// TIA Portal V16 export
// export: Created 2021-11-12T13:32:04.0416234Z, ExportSetting WithDefaults, DisplayName Totally Integrated Automation Portal, DisplayVersion V16 Update 3, DisplayName TIA Portal Version Control Interface, DisplayVersion V16 Update 2, DisplayName TIA Portal Openness, DisplayVersion V16 Update 3, DisplayName SINAMICS Startdrive Advanced, DisplayVersion V16 Update 5, DisplayName SINAMICS Startdrive G130, G150, S120, S150, SINAMICS MV, S210, DisplayVersion V16 Update 5, DisplayName SINAMICS Startdrive G110M, G120, G120C, G120D, G120P, G115D, DisplayVersion V16 Update 5, DisplayName STEP 7 Professional, DisplayVersion V16 Update 3, DisplayName STEP 7 Safety, DisplayVersion V16, DisplayName WinCC UA Professional, DisplayVersion V16 Update 3
DATA_BLOCK "IDB_Station110"   // DB202
VERSION : 0.1
// stored: AutoNumber true, DBAccessibleFromOPCUA true, InstanceOfName Station 110, InstanceOfType FB
"Station 110"
   // VAR
   //    SF_Alarm1 : "STD_DI_Mon";
   //    SF_Alarm2 { S7_SetPoint := 'True'} : "STD_DI_Mon";
   //    SF_Alarm3 { S7_SetPoint := 'True'} : "STD_DI_Mon";
   //    SF_Alarm4 { S7_SetPoint := 'True'} : "STD_DI_Mon";
   //    SF_Alarm5 { S7_SetPoint := 'True'} : "STD_DI_Mon";
   //    SF_Alarm6 { S7_SetPoint := 'True'} : "STD_DI_Mon";
   //    SF_Alarm7 { S7_SetPoint := 'True'} : "STD_DI_Mon";
   //    SF_Alarm8 { S7_SetPoint := 'True'} : "STD_DI_Mon";
   //    SF_Alarm9 { S7_SetPoint := 'True'} : "STD_DI_Mon";
   //    SF_Alarm10 { S7_SetPoint := 'True'} : "STD_DI_Mon";
   //    SF_Alarm11 { S7_SetPoint := 'True'} : "STD_DI_Mon";
   //    SF_Alarm12 { S7_SetPoint := 'True'} : "STD_DI_Mon";
   //    SF_Alarm13 { S7_SetPoint := 'True'} : "STD_DI_Mon";
   //    SF_Alarm14 { S7_SetPoint := 'True'} : "STD_DI_Mon";
   //    SF_Alarm15 { S7_SetPoint := 'True'} : "STD_DI_Mon";
   //    SF_Alarm16 { S7_SetPoint := 'True'} : "STD_DI_Mon";
   //    SF_Alarm17 { S7_SetPoint := 'True'} : "STD_DI_Mon";
   //    SF_Alarm18 { S7_SetPoint := 'True'} : "STD_DI_Mon";
   //    SF_Alarm19 { S7_SetPoint := 'True'} : "STD_DI_Mon";
   //    SF_Alarm20 { S7_SetPoint := 'True'} : "STD_DI_Mon";
   //    SF_Alarm21 { S7_SetPoint := 'True'} : "STD_DI_Mon";
   //    SF_GL01MA02 { S7_SetPoint := 'True'} : "STD_Drive1";
   //    SF_UH31TA01 { S7_SetPoint := 'True'} : "STD_SERVO_FESTO_CMMT";
   //    SF_UC12TA01 { S7_SetPoint := 'True'} : "STD_Siemens_G120_CU240E_2_PN";
   //    SF_GL01BG05 { S7_SetPoint := 'True'} : "STD_Siemens_MC_Encoder";
   //    SF_GL01MM01 { S7_SetPoint := 'True'} : "STD_Valve2WB";
   //    SF_GM01MM01 { S7_SetPoint := 'True'} : "STD_Valve2WB";
   //    SF_GM01MM02 { S7_SetPoint := 'True'} : "STD_Valve2WB";
   //    SF_GM01MM03 { S7_SetPoint := 'True'} : "STD_Valve2WB";
   //    SF_GM01MM04 { S7_SetPoint := 'True'} : "STD_Valve2WB";
   //    SS_Edge : Array[0..9] of Bool;
   //    SF_TON_MeasDelay { S7_SetPoint := 'True'} : TON_TIME;
   //    SR_ConvActPos : Real;
   // END_VAR
   // VAR RETAIN
   //    SR_ConvStopPos : Real;
   //    SB1ConvInPos { ExternalAccessible := 'False'; ExternalVisible := 'False'; ExternalWritable := 'False'} : Bool;
   //    SB1ConvStep : Bool;
   //    SI_SeqStepNr : UInt;
   //    SR_UH31TA01SetPos { ExternalAccessible := 'False'; ExternalVisible := 'False'; ExternalWritable := 'False'} : Real;
   // END_VAR
   // VAR
   //    SR_MeasuredPartLenght : Real;
   //    SI_PartType : Int;
   //    SDIPartID : DInt;
   // END_VAR
BEGIN
END_DATA_BLOCK
